// TwinCAT 3 PLC project tcl_StringUtils
// Title: tcl_StringUtils
// Company: Red Rock Controls Limited
// Author: Roger Christopher
// ProjectVersion: 1.1.7.0
// Description: StringSplitterEx added - strips multiple delimitters.
// ProgramVersion: 3.1.4024.0
// libraries:
//   Tc2_Standard, * (Beckhoff Automation GmbH)
//   Tc2_System, * (Beckhoff Automation GmbH)
//   Tc2_Utilities, * (Beckhoff Automation GmbH)
//   Tc3_Module, * (Beckhoff Automation GmbH)
//   tcl_UnitTestLibrary, * (Red Rock Controls Limited)
// project tree:
//   Classes/ T_LongString.TcPOU, T_StringSplitter.TcPOU, T_StringSplitterEx.TcPOU
//   Functions/Conversion/ F_String_To_IPv4_Address.TcPOU, F_ULINT_TO_TIMESTRUCT.TcPOU, F_TypeClassToString.TcPOU
//   Functions/Date Time Formatting/ F_DateAsString.TcPOU (not stored), F_DateTimeAsString.TcPOU (not stored), F_DateTimeAsString_ms.TcPOU, F_TimeAsString.TcPOU (not stored), F_TimeAsString_ms.TcPOU (not stored), F_TimestampAsFilenameString.TcPOU, F_TimestampAsFilenameString_ms.TcPOU
//   Functions/String Formatting/ F_FormatString1.TcPOU (not stored), F_FormatString10.TcPOU (not stored), F_FormatString2.TcPOU (not stored), F_FormatString3.TcPOU, F_FormatString4.TcPOU, F_FormatString5.TcPOU (not stored), F_FormatString6.TcPOU, F_FormatString7.TcPOU (not stored), F_FormatString8.TcPOU (not stored), F_FormatStringEx1.TcPOU (not stored), F_FormatStringEx10.TcPOU (not stored), F_FormatStringEx2.TcPOU (not stored), F_FormatStringEx3.TcPOU (not stored), F_FormatStringEx4.TcPOU (not stored), F_FormatStringEx5.TcPOU, F_FormatStringEx6.TcPOU (not stored), F_FormatStringEx7.TcPOU (not stored), F_FormatStringEx8.TcPOU (not stored), F_LREAL_TO_STRING.TcPOU, F_LTrimEx.TcPOU, F_PadString.TcPOU (not stored), F_RTrimEx.TcPOU, F_STRING_TO_ARG.TcPOU (not stored), F_Trim.TcPOU
//   Functions/Utils/ F_StringLength.TcPOU
//   Version/ Global_Version.TcGVL
// real-time tasks:
//   TASK PlcTask: cycle T#10ms, priority 1, ADS port 350

// ---- Version/Global_Version.TcGVL
{attribute 'TcGenerated'}
{attribute 'no-analysis'}
{attribute 'linkalways'}
// This function has been automatically generated from the project information.
VAR_GLOBAL CONSTANT
	{attribute 'const_non_replaced'}
	stLibVersion_tcl_StringUtils : ST_LibVersion := (iMajor := 1, iMinor := 1, iBuild := 7, iRevision := 0, nFlags := 0, sVersion := '1.1.7.0');
END_VAR

// ---- Classes/T_LongString.TcPOU
FUNCTION_BLOCK T_LongString
VAR
    buffer : STRING(MAX_LENGTH);
    CharCount : UDINT;
END_VAR
VAR CONSTANT
    MAX_LENGTH : UDINT := 1024;
END_VAR

PROPERTY Address : PVOID
GET
Address := ADR(Buffer);
END_GET
END_PROPERTY

METHOD AppendString
VAR_INPUT
    str : T_MaxString;
END_VAR
VAR
    stringLength : UDINT;
END_VAR
stringLength := INT_TO_UDINT(LEN(str));

IF (stringLength + CharCount < MAX_LENGTH - 1) THEN
    MEMCPY(
        destAddr := Address + CharCount,
        srcAddr  := ADR(str),
        n        := stringLength);
    CharCount := CharCount + stringLength;       
END_IF
END_METHOD

METHOD Clear
VAR_INPUT
END_VAR
MEMSET(Address,0,MAX_LENGTH);
CharCount := 0;
END_METHOD

PROPERTY Length : UDINT
GET
Length := CharCount;
END_GET
END_PROPERTY

END_FUNCTION_BLOCK

// ---- Classes/T_StringSplitter.TcPOU
FUNCTION_BLOCK T_StringSplitter
VAR
	SubjectString : TC2_SYSTEM.T_MaxString;
	Delimiter : STRING;
	Delimiter1 : STRING;
	Delimiter2 : STRING;
	NextDelimiterPosition : INT;
	NextDelimiter1Position : INT;
	NextDelimiter2Position : INT;
END_VAR

METHOD GetNext : STRING(255)
VAR_INPUT
END_VAR
VAR
	RemainingLength: INT;
END_VAR
NextDelimiter1Position := FIND(SubjectString , Delimiter1);
NextDelimiter2Position := FIND(SubjectString , Delimiter2);

IF NextDelimiter1Position = 0 THEN
    // use Delimiter 2 position , even if zero...
    NextDelimiterPosition := NextDelimiter2Position;
    Delimiter := Delimiter2;
    
ELSIF NextDelimiter2Position = 0 THEN
    // use Delimiter 1 position , non-zero...
    NextDelimiterPosition := NextDelimiter1Position;
    Delimiter := Delimiter1;

ELSE
    // Both delimters found - use the one nearest the start of the string...
    IF NextDelimiter1Position < NextDelimiter2Position THEN
        NextDelimiterPosition := NextDelimiter1Position;
        Delimiter := Delimiter1;
    ELSE
        NextDelimiterPosition := NextDelimiter2Position;
        Delimiter := Delimiter2;
	END_IF
END_IF

IF NextDelimiterPosition > 0 THEN // delimitter found
    
    // extract next sub-string
	GetNext := LEFT(SubjectString,NextDelimiterPosition - 1);
    
    // remove sub-string from subject string
	RemainingLength := LEN(SubjectString) - NextDelimiterPosition - LEN(Delimiter) + 1;
	SubjectString := RIGHT(SubjectString,RemainingLength);
    
//    // strip any delimitters from front of remaining string
//    WHILE FIND(SubjectString,Delimiter1) = 1 DO
//        SubjectString := RIGHT(SubjectString,LEN(SubjectString) - LEN(Delimiter1));
//	END_WHILE
//    WHILE FIND(SubjectString,Delimiter2) = 1 DO
//        SubjectString := RIGHT(SubjectString,LEN(SubjectString) - LEN(Delimiter2));
//	END_WHILE
ELSE
	GetNext := SubjectString; // return what is left
	SubjectString := '';
END_IF
END_METHOD

METHOD GetRemainder : STRING(255)
GetRemainder := SubjectString; // return what is left
SubjectString := '';
END_METHOD

METHOD HasMore : BOOL
VAR_INPUT
END_VAR
HasMore := SubjectString <> '';
END_METHOD

METHOD Init
VAR_INPUT
		Str : TC2_SYSTEM.T_MaxString;
		Delim1 : STRING;
		Delim2 : STRING;
END_VAR
SubjectString := Str;
NextDelimiterPosition := 0;
Delimiter1 := Delim1;
Delimiter2 := Delim2;
END_METHOD

END_FUNCTION_BLOCK

// ---- Classes/T_StringSplitterEx.TcPOU
FUNCTION_BLOCK T_StringSplitterEx
VAR
	SubjectString : TC2_SYSTEM.T_MaxString;
	Delimiter : STRING;
	Delimiter1 : STRING;
	Delimiter2 : STRING;
	NextDelimiterPosition : INT;
	NextDelimiter1Position : INT;
	NextDelimiter2Position : INT;
END_VAR

METHOD GetNext : STRING(255)
VAR_INPUT
END_VAR
VAR
	RemainingLength: INT;
END_VAR
NextDelimiter1Position := FIND(SubjectString , Delimiter1);
NextDelimiter2Position := FIND(SubjectString , Delimiter2);

IF NextDelimiter1Position = 0 THEN
    // use Delimiter 2 position , even if zero...
    NextDelimiterPosition := NextDelimiter2Position;
    Delimiter := Delimiter2;
    
ELSIF NextDelimiter2Position = 0 THEN
    // use Delimiter 1 position , non-zero...
    NextDelimiterPosition := NextDelimiter1Position;
    Delimiter := Delimiter1;

ELSE
    // Both delimters found - use the one nearest the start of the string...
    IF NextDelimiter1Position < NextDelimiter2Position THEN
        NextDelimiterPosition := NextDelimiter1Position;
        Delimiter := Delimiter1;
    ELSE
        NextDelimiterPosition := NextDelimiter2Position;
        Delimiter := Delimiter2;
	END_IF
END_IF

IF NextDelimiterPosition > 0 THEN // delimitter found
    
    // extract next sub-string
	GetNext := LEFT(SubjectString,NextDelimiterPosition - 1);
    
    // remove sub-string from subject string
	RemainingLength := LEN(SubjectString) - NextDelimiterPosition - LEN(Delimiter) + 1;
	SubjectString := RIGHT(SubjectString,RemainingLength);
    
    // strip any delimitters from front of remaining string
    WHILE FIND(SubjectString,Delimiter1) = 1 DO
        SubjectString := RIGHT(SubjectString,LEN(SubjectString) - LEN(Delimiter1));
	END_WHILE
    WHILE FIND(SubjectString,Delimiter2) = 1 DO
        SubjectString := RIGHT(SubjectString,LEN(SubjectString) - LEN(Delimiter2));
	END_WHILE
	
ELSE
	GetNext := SubjectString; // return what is left
	SubjectString := '';
END_IF
END_METHOD

METHOD GetRemainder : STRING(255)
GetRemainder := SubjectString; // return what is left
SubjectString := '';
END_METHOD

METHOD HasMore : BOOL
VAR_INPUT
END_VAR
HasMore := SubjectString <> '';
END_METHOD

METHOD Init
VAR_INPUT
		Str : TC2_SYSTEM.T_MaxString;
		Delim1 : STRING;
		Delim2 : STRING;
END_VAR
SubjectString := Str;
NextDelimiterPosition := 0;
Delimiter1 := Delim1;
Delimiter2 := Delim2;
END_METHOD

END_FUNCTION_BLOCK

// ---- Functions/Conversion/F_String_To_IPv4_Address.TcPOU
FUNCTION F_String_To_IPv4_Address : ARRAY[1..4] of BYTE
VAR_INPUT
    IpAddress : STRING; // like 192.168.1.125
END_VAR
VAR
    StringSplitter : T_StringSplitter;
    Byte1          : STRING;
    Byte2          : STRING;
    Byte3          : STRING;
    Byte4          : STRING;
    Result         : ARRAY[1..4] OF BYTE;
END_VAR

StringSplitter.Init(IpAddress,
                    '.',
                    '');

Byte4 := StringSplitter.GetNext();
Byte3 := StringSplitter.GetNext();
Byte2 := StringSplitter.GetNext();
Byte1 := StringSplitter.GetNext();

Result[1] := STRING_TO_BYTE(Byte1);
Result[2] := STRING_TO_BYTE(Byte2);
Result[3] := STRING_TO_BYTE(Byte3);
Result[4] := STRING_TO_BYTE(Byte4);

F_String_To_IPv4_Address := Result;

END_FUNCTION

// ---- Functions/Conversion/F_ULINT_TO_TIMESTRUCT.TcPOU
FUNCTION F_ULINT_TO_TIMESTRUCT : TIMESTRUCT
VAR_INPUT
	TimeStamp : ULINT; // data type og eventLogger3 timestamp - number of 100nS since 1601
END_VAR
VAR
	pFileTime : POINTER TO T_FILETIME;
	Result : TIMESTRUCT;
END_VAR

pFileTime := ADR(TimeStamp);
Result := FILETIME_TO_SYSTEMTIME(pFileTime^);

F_ULINT_TO_TIMESTRUCT := Result;

END_FUNCTION

// ---- Functions/Conversion/F_TypeClassToString.TcPOU
FUNCTION F_TypeClassToString : STRING
VAR_INPUT
    TypeClass : __SYSTEM.TYPE_CLASS;
END_VAR
VAR
    Result : STRING;
END_VAR

CASE TypeClass OF
    __SYSTEM.TYPE_CLASS.TYPE_BOOL          : Result := 'BOOL';
    __SYSTEM.TYPE_CLASS.TYPE_BIT           : Result := 'BOOL';
    __SYSTEM.TYPE_CLASS.TYPE_BYTE          : Result := 'BYTE';
    __SYSTEM.TYPE_CLASS.TYPE_WORD          : Result := 'WORD';
    __SYSTEM.TYPE_CLASS.TYPE_DWORD         : Result := 'DWORD';
    __SYSTEM.TYPE_CLASS.TYPE_LWORD         : Result := 'DWORD';
    __SYSTEM.TYPE_CLASS.TYPE_SINT          : Result := 'SINT';
    __SYSTEM.TYPE_CLASS.TYPE_INT           : Result := 'INT';
    __SYSTEM.TYPE_CLASS.TYPE_DINT          : Result := 'DINT';
    __SYSTEM.TYPE_CLASS.TYPE_LINT          : Result := 'LINT';
    __SYSTEM.TYPE_CLASS.TYPE_USINT         : Result := 'USINT';
    __SYSTEM.TYPE_CLASS.TYPE_UINT          : Result := 'UINT';
    __SYSTEM.TYPE_CLASS.TYPE_UDINT         : Result := 'UDINT';
    __SYSTEM.TYPE_CLASS.TYPE_ULINT         : Result := 'ULINT';
    __SYSTEM.TYPE_CLASS.TYPE_REAL          : Result := 'REAL';
    __SYSTEM.TYPE_CLASS.TYPE_LREAL         : Result := 'LREAL';
    __SYSTEM.TYPE_CLASS.TYPE_STRING        : Result := 'STRING';
    __SYSTEM.TYPE_CLASS.TYPE_WSTRING       : Result := 'WSTRING';     
    __SYSTEM.TYPE_CLASS.TYPE_TIME          : Result := 'TIME';        
    __SYSTEM.TYPE_CLASS.TYPE_DATE          : Result := 'DATE';        
    __SYSTEM.TYPE_CLASS.TYPE_DATEANDTIME   : Result := 'DATEANDTIME'; 
    __SYSTEM.TYPE_CLASS.TYPE_TIMEOFDAY     : Result := 'TIMEOFDAY';   
    __SYSTEM.TYPE_CLASS.TYPE_POINTER       : Result := 'POINTER';     
    __SYSTEM.TYPE_CLASS.TYPE_REFERENCE     : Result := 'REFERENCE';   
    __SYSTEM.TYPE_CLASS.TYPE_SUBRANGE      : Result := 'SUBRANGE';    
    __SYSTEM.TYPE_CLASS.TYPE_ENUM          : Result := 'ENUM';        
    __SYSTEM.TYPE_CLASS.TYPE_ARRAY         : Result := 'ARRAY';      
    __SYSTEM.TYPE_CLASS.TYPE_PARAMS        : Result := 'PARAMS';      
    __SYSTEM.TYPE_CLASS.TYPE_USERDEF       : Result := 'USERDEF';     
    __SYSTEM.TYPE_CLASS.TYPE_NONE          : Result := 'NONE';        
    __SYSTEM.TYPE_CLASS.TYPE_ANY           : Result := 'ANY';         
    __SYSTEM.TYPE_CLASS.TYPE_ANYBIT        : Result := 'ANYBIT';      
    __SYSTEM.TYPE_CLASS.TYPE_ANYDATE       : Result := 'ANYDATE';     
    __SYSTEM.TYPE_CLASS.TYPE_ANYINT        : Result := 'ANYINT';      
    __SYSTEM.TYPE_CLASS.TYPE_ANYNUM        : Result := 'ANYNUM';      
    __SYSTEM.TYPE_CLASS.TYPE_ANYREAL       : Result := 'ANYREAL';     
    __SYSTEM.TYPE_CLASS.TYPE_LAZY          : Result := 'LAZY';        
    __SYSTEM.TYPE_CLASS.TYPE_BITCONST      : Result := 'BITCONST';    
ELSE
    Result := DWORD_TO_STRING(TypeClass);
END_CASE

F_TypeClassToString := Result;

END_FUNCTION

// ---- Functions/Date Time Formatting/F_DateTimeAsString_ms.TcPOU
FUNCTION F_DateTimeAsString_ms : T_MaxString
VAR_INPUT
    TimeStruct : TIMESTRUCT;
END_VAR

F_DateTimeAsString_ms := F_FormatStringEx2(
                             Format := '%s %s',
                             arg1   := F_TimeAsString_ms(TimeStruct),
                             arg2   := F_DateAsString(TimeStruct));

END_FUNCTION

// ---- Functions/Date Time Formatting/F_TimestampAsFilenameString.TcPOU
FUNCTION F_TimestampAsFilenameString : T_MaxString
VAR_INPUT
    TimeStruct : TIMESTRUCT;
END_VAR
VAR
	FB_FormatString1 : FB_FormatString;
END_VAR

FB_FormatString1(
	sFormat:= '%.2d-%.2d-%.2d %.2d-%.2d-%.2d', 
	arg1:= F_WORD(TimeStruct.wYear), 
	arg2:= F_WORD(TimeStruct.wMonth), 
	arg3:= F_WORD(TimeStruct.wDay),
	arg4:= F_WORD(TimeStruct.wHour),
	arg5:= F_WORD(TimeStruct.wMinute), 
	arg6:= F_WORD(TimeStruct.wSecond), 
	arg7:= ,
	arg8:= , 
	arg9:= , 
	arg10:= , 
	bError=> , 
	nErrId=> , 
	sOut=> F_TimestampAsFilenameString);

END_FUNCTION

// ---- Functions/Date Time Formatting/F_TimestampAsFilenameString_ms.TcPOU
FUNCTION F_TimestampAsFilenameString_ms : T_MaxString
VAR_INPUT
    TimeStruct : TIMESTRUCT;
END_VAR
VAR
	FB_FormatString1 : FB_FormatString;
END_VAR

FB_FormatString1(
	sFormat:= '%.2d-%.2d-%.2d %.2d:%.2d:%.2d.%.3d', 
	arg1:= F_WORD(TimeStruct.wYear), 
	arg2:= F_WORD(TimeStruct.wMonth), 
	arg3:= F_WORD(TimeStruct.wDay),
	arg4:= F_WORD(TimeStruct.wHour),
	arg5:= F_WORD(TimeStruct.wMinute), 
	arg6:= F_WORD(TimeStruct.wSecond), 
	arg7:= F_WORD(TimeStruct.wMilliseconds),
	arg8:= , 
	arg9:= , 
	arg10:= , 
	bError=> , 
	nErrId=> , 
	sOut=> F_TimestampAsFilenameString_ms);

END_FUNCTION

// ---- Functions/String Formatting/F_FormatString3.TcPOU
FUNCTION F_FormatString3 : T_MaxString
VAR_INPUT
	Format	: T_MaxString;
	arg1	: T_Arg;
	arg2	: T_Arg;
	arg3	: T_Arg;
END_VAR
VAR
    FB_FormatString1 : FB_FormatString;
END_VAR

FB_FormatString1(
	sFormat:= Format, 
	arg1:= arg1, 
	arg2:= arg2, 
	arg3:= arg3, 
	arg4:= , 
	arg5:= , 
	arg6:= , 
	arg7:= , 
	arg8:= , 
	arg9:= , 
	arg10:= , 
	bError=> , 
	nErrId=> , 
	sOut=> F_FormatString3);

END_FUNCTION

// ---- Functions/String Formatting/F_FormatString4.TcPOU
FUNCTION F_FormatString4 : T_MaxString
VAR_INPUT
	Format	: T_MaxString;
	arg1	: T_Arg;
	arg2	: T_Arg;
	arg3	: T_Arg;
	arg4	: T_Arg;
END_VAR
VAR
    FB_FormatString1 : FB_FormatString;
END_VAR

FB_FormatString1(
	sFormat:= Format, 
	arg1:= arg1, 
	arg2:= arg2, 
	arg3:= arg3, 
	arg4:= arg4, 
	arg5:= , 
	arg6:= , 
	arg7:= , 
	arg8:= , 
	arg9:= , 
	arg10:= , 
	bError=> , 
	nErrId=> , 
	sOut=> F_FormatString4);

END_FUNCTION

// ---- Functions/String Formatting/F_FormatString6.TcPOU
FUNCTION F_FormatString6 : T_MaxString
VAR_INPUT
	Format	: T_MaxString;
	arg1	: T_Arg;
	arg2	: T_Arg;
	arg3	: T_Arg;
	arg4	: T_Arg;
	arg5	: T_Arg;
	arg6	: T_Arg;
END_VAR
VAR
    FB_FormatString1 : FB_FormatString;
END_VAR

FB_FormatString1(
	sFormat:= Format, 
	arg1:= arg1, 
	arg2:= arg2, 
	arg3:= arg3, 
	arg4:= arg4, 
	arg5:= arg5, 
	arg6:= arg6, 
	arg7:= , 
	arg8:= , 
	arg9:= , 
	arg10:= , 
	bError=> , 
	nErrId=> , 
	sOut=> F_FormatString6);

END_FUNCTION

// ---- Functions/String Formatting/F_FormatStringEx5.TcPOU
FUNCTION F_FormatStringEx5 : T_MaxString
VAR_INPUT
	Format	: T_MaxString;
	arg1	: T_MaxString;
	arg2	: T_MaxString;
	arg3	: T_MaxString;
	arg4	: T_MaxString;
	arg5	: T_MaxString;
END_VAR
VAR
    FB_FormatString1 : FB_FormatString;
END_VAR



FB_FormatString1(
	sFormat:= Format, 
	arg1:= F_STRING(arg1), 
	arg2:= F_STRING(arg2),
	arg3:= F_STRING(arg3), 
	arg4:= F_STRING(arg4), 
	arg5:= F_STRING(arg5), 
	arg6:= , 
	arg7:= , 
	arg8:= , 
	arg9:= , 
	arg10:= , 
	bError=> , 
	nErrId=> , 
	sOut=> F_FormatStringEx5);

END_FUNCTION

// ---- Functions/String Formatting/F_LREAL_TO_STRING.TcPOU
FUNCTION F_LREAL_TO_STRING : STRING
VAR_INPUT
    Value : LREAL;
    Precision : INT;
END_VAR
VAR
END_VAR

F_LREAL_TO_STRING := LREAL_TO_FMTSTR(in := Value,
                                     iPrecision := Precision,
                                     bRound := TRUE);

END_FUNCTION

// ---- Functions/String Formatting/F_LTrimEx.TcPOU
FUNCTION F_LTrimEx : T_MaxString // removes n characters from start of string
VAR_INPUT
   n : UINT; 
   str : T_MaxString;
END_VAR
VAR
    Length : UINT;
END_VAR

Length := INT_TO_UINT(LEN(str));
IF n = 0 THEN
    F_LTrimEx := str;
ELSIF n < Length THEN
    MEMCPY(destAddr := ADR(F_LTrimEx),
           srcAddr  := ADR(str) + n,
           n        := Length - n + 1); // include null terminator
ELSE
	F_LTrimEx := ''; // remove everything
END_IF

END_FUNCTION

// ---- Functions/String Formatting/F_RTrimEx.TcPOU
FUNCTION F_RTrimEx : T_MaxString // removes n characters from end of string
VAR_INPUT
   n : UINT; 
   str : T_MaxString;
END_VAR
VAR
    Length : UINT;
END_VAR

Length := INT_TO_UINT(LEN(str));
IF n = 0 THEN
    F_RTrimEx := str;
ELSIF n < Length THEN
    // overwrite chars to be trimmed with nulls...
    MEMSET(destAddr := ADR(str) + Length - n,
           fillByte:= 0,
           n := n); 
	F_RTrimEx := str;
ELSE
	F_RTrimEx := ''; // remove everything
END_IF

END_FUNCTION

// ---- Functions/String Formatting/F_Trim.TcPOU
FUNCTION F_Trim : T_MaxString
VAR_INPUT
	str: T_MaxString;
END_VAR
VAR
	Result: T_MaxString;
END_VAR

Result := str;
WHILE 
    LEFT(Result,1) = '$T'
OR 
    LEFT(Result,1) = ' '
DO
	Result := F_LTrimEx(n := 1, str := Result); // Strip tabs and spaces from LHS
END_WHILE

WHILE 
    RIGHT(Result,1) = '$R'
OR 
    RIGHT(Result,1) = '$N'
OR 
    RIGHT(Result,1) = '$T'
OR 
    RIGHT(Result,1) = ' '
DO
	Result := F_RTrimEx(n := 1, str := Result); // Strip tabs, Spaces, CR and LF from RHS
END_WHILE


F_Trim := Result;

END_FUNCTION

// ---- Functions/Utils/F_StringLength.TcPOU
FUNCTION F_StringLength : UDINT
VAR_IN_OUT CONSTANT
	str : STRING;
END_VAR
VAR
	pByte : POINTER TO BYTE;
END_VAR

pByte := ADR(str);

WHILE pByte^ <> 0 DO
	pByte := pByte + 1;
	F_StringLength := F_StringLength + 1;
END_WHILE

END_FUNCTION
